FUNCTION_BLOCK FB_Diverter_Module001 EXTENDS FB_PackML_BaseModule
VAR
	// Sub module definitions here

	// List of sub modules
	ipSubModules_Init : ARRAY[1..Parameters_PackML_Base.MAX_NO_OF_SUBMODULES] OF I_PackML_BaseModule := [];

	// Component definitions here
//	Axis   : FB_Component_BasicAxis := (Name := 'Axis');
	Drive_1	:I_Drive_Type_1_Axis;
	Drive_2	:I_Drive_Type_1_Axis;
	Sensor : FB_DigitalSensor		:= (Name := 'Sensor');

	//Alarms for this module
	DiverterAlarms : ARRAY[1..DIVERTER_ALARM_COUNT] OF FB_TcAlarm;

	//Data for recipe
	Recipe : ST_DiverterRecipe;

	(*Parameters from PackTags for module
    //_Param  : ARRAY[1..10] OF ST_Descriptor2;*)
	_Report : ARRAY[1..10] OF ST_Descriptor2;

	//HMI Control for EM
	fbControlSourceHMI : FB_ControlSource_HMI;
END_VAR

VAR CONSTANT
	//reports 
	FAULT : INT := 1;

	//Alarms
	DIVERTER_ALARM_COUNT : INT := 5;
END_VAR

//Simulation variables for messaging
VAR
	ErrorInput : BOOL;
	WarnInput  : BOOL;
	InfoInput  : BOOL;
END_VAR

METHOD PROTECTED Aborting
VAR_INPUT
END_VAR
CASE SequenceState OF
	0:
		NoStateTasksToComplete := FALSE;
		SequenceState		   := SequenceState + 10;

	10:
	//	Axis.Stop();
	//	IF Axis.Stopped THEN
			SequenceState := SequenceState + 10;
	//	END_IF

	20:
		// Disable here
	//	Axis.Disable();

		// Check not enabled here
	//	IF NOT Axis.Enabled THEN
			SequenceState := SequenceState + 10;
	//	END_IF

	30:
		StateTasksComplete := TRUE;
END_CASE

SUPER^.Aborting();
END_METHOD

PROPERTY Acceleration : LREAL
SET
//Recipe.Axis.Acceleration := Acceleration;
END_SET
END_PROPERTY

METHOD PROTECTED Clearing
VAR_INPUT
END_VAR
CASE SequenceState OF
	0:
		NoStateTasksToComplete := FALSE;
		SequenceState		   := SequenceState + 10;

	10:
		//Reset any alarms that get latched
		DiverterAlarms[E_Unwind.StartTimeout].Clear(0, 0);
		SequenceState := SequenceState + 10;

	20:
		// Enable here
	//	Axis.Enable();

		// Check enabled here
	//	IF Axis.Enabled THEN
			SequenceState := SequenceState + 10;
	//	END_IF

	30:
		StateTasksComplete := TRUE;
END_CASE

SUPER^.Clearing();
END_METHOD

METHOD PROTECTED CreateEvents
VAR_INPUT
END_VAR
// Add your event creation here
F_CreateAllEventsInClass(Alarms		:= DiverterAlarms,
						 ClassSize	:= SIZEOF(TC_EVENTS.Unwind),
						 pInitEvent := ADR(TC_EVENTS.Unwind.InitReferenceEvent),
						 Prefix		:= Name);

// Super call to base
SUPER^.CreateEvents();
END_METHOD

METHOD CyclicLogic
VAR_INPUT
END_VAR
IF NOT _InitComplete THEN
	_InitComplete := Initialize();
	RETURN;
END_IF

SUPER^.CyclicLogic();

//HMI control for EM
fbControlSourceHMI.CyclicLogic();

//Set the current alarm severity for this module
_CurrentAlarmSeverity := F_GetMaxSeverityRaised(Alarms := DiverterAlarms, CurrentSeverity := _CurrentAlarmSeverity);
IF _CurrentAlarmSeverity >= TcEventSeverity.Error THEN
	ChangeState(E_PMLCommand.ePMLCommand_Abort);
END_IF

//CyclicLogic_Simulation();
END_METHOD

METHOD CyclicLogic_Simulation
VAR_INPUT
END_VAR
(*	
This is just for testing. Real hardware can be setup in other places
Here the alarms will raise and clear on its own if the input changes	
*)

//Generic Alarms for Testing
IF ErrorInput AND NOT UnwindAlarms[E_Unwind.AlarmMessage].bRaised THEN
	RaiseAlarm2Args(UnwindAlarms[E_Unwind.AlarmMessage], '', '');
ELSIF NOT ErrorInput AND UnwindAlarms[E_Unwind.AlarmMessage].bRaised THEN
	UnwindAlarms[E_Unwind.AlarmMessage].Clear(0, 0);
END_IF

IF WarnInput AND NOT UnwindAlarms[E_Unwind.WarnMessage].bRaised THEN
	RaiseAlarm2Args(UnwindAlarms[E_Unwind.WarnMessage], '', '');
ELSIF NOT WarnInput AND UnwindAlarms[E_Unwind.WarnMessage].bRaised THEN
	UnwindAlarms[E_Unwind.WarnMessage].Clear(0, 0);
END_IF

IF InfoInput AND NOT UnwindAlarms[E_Unwind.InfoMessage].bRaised THEN
	RaiseAlarm2Args(UnwindAlarms[E_Unwind.InfoMessage], '', '');
ELSIF NOT InfoInput AND UnwindAlarms[E_Unwind.InfoMessage].bRaised THEN
	UnwindAlarms[E_Unwind.InfoMessage].Clear(0, 0);
END_IF
END_METHOD

METHOD FB_init : BOOL
VAR_INPUT
	bInitRetains : BOOL; // if TRUE, the retain variables are initialized (warm start / cold start)
	bInCopyCode : BOOL;  // if TRUE, the instance afterwards gets moved into the copy code (online change)
	Drive_1	:I_Drive_Type_1_Axis;
	Drive_2	:I_Drive_Type_1_Axis;
END_VAR
THIS^.Drive_1	:=	Drive_1 ;
THIS^.Drive_2	:=	Drive_2 ;
END_METHOD

//! @summary Basic module initialization logic
METHOD PROTECTED Initialize : BOOL;
VAR
	i						 : UDINT;
	varInfo					 : __SYSTEM.VAR_INFO;
	AllSubUnitsInitialized	 : BOOL := TRUE;
	AllComponentsInitialized : BOOL := TRUE;
END_VAR

//! @description This method is called by <c>CyclicLogic()</c> as required
Initialize := FALSE;
CASE DescendantSequenceState OF
	0:
	//	RegisterComponent(Axis);
	//	RegisterComponent(Drive_1);
		RegisterComponent(Sensor);
		_LogModeChanges			:= FALSE;
		_LogStateChanges		:= FALSE;
		DescendantSequenceState := DescendantSequenceState + 10;

	10:
		//Setup Custom modes here

		(*CustomModes(eMode                          :=,
                    sName                          :=,
                    bDisableClearing               :=,
                    bDisableStarting               :=,
                    bDisableSuspended              :=,
                    bDisableStopping               :=,
                    bDisableAborting               :=,
                    bDisableHolding                :=,
                    bDisableHeld                   :=,
                    bDisableUnholding              :=,
                    bDisableSuspending             :=,
                    bDisableUnsuspending           :=,
                    bDisableResetting              :=,
                    bDisableIdle                   :=,
                    bDisableCompleting             :=,
                    bDisableComplete               :=,
                    bEnableUnitModeChangeStopped   :=,
                    bEnableUnitModeChangeIdle      :=,
                    bEnableUnitModeChangeSuspended :=,
                    bEnableUnitModeChangeExecute   :=,
                    bEnableUnitModeChangeAborted   :=,
                    bEnableUnitModeChangeHeld      :=,
                    bEnableUnitModeChangeComplete  :=,
                    bError                         =>,
                    nErrorId                       =>);*)
		DescendantSequenceState := DescendantSequenceState + 10;

	20:
		//Copy Mode names
		FOR i := 1 TO 3 DO
			ModeNames[i] := F_UnitModeToString(UDINT_TO_DINT(i));
		END_FOR

		Initialize_TagData();
		RegisterExternalController(Controller := fbControlSourceHMI);
		fbControlSourceHMI.CyclicLogic();

		//Set the Parent Response here
		_ParentFaultResponseDefinitions[TcEventSeverity.Error] := E_AlarmResponse.Hold_Immediate;
		DescendantSequenceState								   := DescendantSequenceState + 10;

	30:
		//Call the Super
		IF SUPER^.Initialize() THEN
			DescendantSequenceState := DescendantSequenceState + 10;
		END_IF

	40:
		Initialize := TRUE;
END_CASE
END_METHOD

METHOD Initialize_TagData
VAR_INPUT
END_VAR
//Recipe
//Recipe.Axis.Velocity	 := 100;
//Recipe.Axis.Acceleration := 1000;

//Report
_Report[FAULT].ID	:= TO_DINT(3 * 10 + 1);
_Report[FAULT].Name := 'Fault ID';
_Report[FAULT].Unit := 'n/a';
END_METHOD

METHOD RaiseAlarm2Args
VAR_IN_OUT
	Alarm : FB_TcAlarm; //Alarm to be raised
END_VAR

VAR_INPUT
	String_1 : STRING; //First String Parameter (The Name of this component will be applied first automatically)
	String_2 : STRING; //Second String Parameter
END_VAR
F_RaiseAlarmWithStringParameters(Alarm	  := Alarm,
								 String_1 := Name,
								 String_2 := String_1,
								 String_3 := String_2);
END_METHOD

METHOD PROTECTED Starting
VAR_INPUT
END_VAR

VAR_INST
	StartTimer : TON;
END_VAR
CASE _CurrentMode OF
	//=================================PRODUCTION MODE==================================
	E_PMLUnitMode.ePMLUnitMode_Production:
		CASE SequenceState OF
			0:
				// Delay 1 scan to make sure timer is off.  Not guarnteed from last time where it finished.
				NoStateTasksToComplete := FALSE;
				SequenceState		   := SequenceState + 10;

			10:
				NoStateTasksToComplete := FALSE;
//				Axis.Velocity		   := Recipe.Axis.Velocity;
//				Axis.Acceleration	   := Recipe.Axis.Acceleration;
//				Axis.MoveVelocity(Velocity := Recipe.Axis.Velocity, AbortPrevious := FALSE);
				SequenceState := SequenceState + 10;

			20:
		//		IF Axis.Busy THEN
					SequenceState := SequenceState + 10;
		//		END_IF

				IF StartTimer.Q AND NOT DiverterAlarms[E_Unwind.StartTimeout].bRaised THEN
					RaiseAlarm2Args(DiverterAlarms[E_Unwind.StartTimeout], '', '');
					SequenceState := SequenceState + 10;
				END_IF

			30:
				StateTasksComplete := TRUE;
		END_CASE

	//=================================MAINTENANCE & MANUAL MODE==================================
	E_PMLUnitMode.ePMLUnitMode_Maintenance, E_PMLUnitMode.ePMLUnitMode_Manual:
		;
END_CASE

SUPER^.Starting();
StartTimer(IN := (SequenceState = 10 OR SequenceState = 20), PT := T#3S);
END_METHOD

METHOD PROTECTED Stopping
VAR_INPUT
END_VAR
CASE _CurrentMode OF
	//=================================PRODUCTION MODE==================================
	E_PMLUnitMode.ePMLUnitMode_Production:
		CASE SequenceState OF
			0:
				NoStateTasksToComplete := FALSE;
		//		Axis.Stop();
				SequenceState := SequenceState + 10;

			10:
		//		IF Axis.Stopped THEN
					SequenceState := SequenceState + 10;
		//		END_IF

			20:
				StateTasksComplete := TRUE;
		END_CASE

	//=================================MAINTENANCE & MANUAL MODE==================================
	E_PMLUnitMode.ePMLUnitMode_Maintenance, E_PMLUnitMode.ePMLUnitMode_Manual:
		;
END_CASE

SUPER^.Stopping();
END_METHOD

PROPERTY Velocity : LREAL
SET
//Recipe.Axis.Velocity := Velocity;
END_SET
END_PROPERTY

END_FUNCTION_BLOCK

(* stored: Version 1.1.0.1, ProductVersion 3.1.4024.15
   POU FB_Diverter_Module001: Id {50568873-dc6a-4c9e-a276-6bb23a8a9804}, SpecialFunc None
   Folder I_CyclicFB: Id {edd6a3fd-60ff-48c2-afaa-993c1d071d27}
   Folder Methods: Id {6166b055-45da-48b7-8f6c-84f1cef16c4d}
   Folder Acting States: Id {f0911c9d-40e9-459e-8a2c-48ab3f313d4a}
   Folder AlarmHandling: Id {bdfad65f-a283-45c1-9036-af466acfd03d}
   Folder Properties: Id {e80a6c7a-b0e5-4900-9835-1415a7875b52}
   Method Aborting: Id {08a648d5-f33e-438b-9f28-2b648e557354}
   Property Acceleration: Id {f3e63590-f71e-48dc-a83b-b01231f47d9a}
   Set Set: Id {ecf2218a-f979-4ab0-8ada-77ed9e94a0f5}
   Method Clearing: Id {8dcd65f3-6e2f-473f-9a4c-ff06653407f6}
   Method CreateEvents: Id {8969e5aa-15f5-445d-8b29-5c7df4d11821}
   Method CyclicLogic: Id {6ab63a94-cb3a-4156-975a-c89c3aef5ba4}
   Method CyclicLogic_Simulation: Id {dbc399a6-4009-48b5-9110-4bc72503ba64}
   Method FB_init: Id {0eef9944-4cd7-45cb-bbff-e395fe038429}
   Method Initialize: Id {025e46ff-9b8a-43d8-9628-052cfbd4f887}
   Method Initialize_TagData: Id {4fb8e91e-c4b4-4e16-a54d-01cf491bcfd5}
   Method RaiseAlarm2Args: Id {4b24d87a-b826-403b-b716-425f76b0b032}
   Method Starting: Id {96425aff-edfb-4aac-8e8a-5b1f8559a712}
   Method Stopping: Id {47895a6f-6ce6-4f2f-8eb3-250f3d1329a5}
   Property Velocity: Id {78058d2b-e6ef-4f0f-a194-31a88871c1ef}
   Set Set: Id {54169eb2-78db-41b8-88a5-dd59bd9e83b1} *)
